// TIA Portal project "Perron038 AMR Siemens" (V14)

(* hardware
DEVICE "S7-1200 station_1"  S7-1200 Station
   slot 0: "Rack_0"  S7-1200 Rack  Rack  V1.0
   slot 1: "PLC_1"  CPU 1215C DC/DC/DC  6ES7 215-1AG40-0XB0  V4.2
*)

// ===== PLC "PLC_1"  CPU 1215C DC/DC/DC =====

VAR_GLOBAL   // PLC tag table "Default tag table"
   "Tag_1" AT %QW1000 : Word;
   "o_Output2" AT %Q0.1 : Bool;
   "Axis_1_Pulse" AT %Q0.0 : Bool;
   "M_stepEnable" AT %I0.0 : Bool;
   "q_driveEn" AT %Q0.2 : Bool;
   "q_stepOff" AT %Q0.3 : Bool;
   "M_ResetAxis" AT %I0.1 : Bool;
   "Jog_For" AT %I0.2 : Bool;
   "Jog_BWD" AT %I0.3 : Bool;
END_VAR

DATA_BLOCK "mainLogic_DB"   // DB1
{ S7_Optimized_Access := 'TRUE' }
VERSION : 0.1
// stored: InstanceOfName mainLogic
"mainLogic"
BEGIN
END_DATA_BLOCK

DATA_BLOCK "Axis_1"   // DB3, Motion_DB
{ S7_Optimized_Access := 'TRUE' }
AUTHOR : SIMATIC
FAMILY : BasicMC
NAME : TO_PosAx
VERSION : 6.0
// stored: InstanceOfName TO_PositioningAxis
"TO_PositioningAxis"
BEGIN
   // Axis.EnableOutput_AddressCU = %Q0.2
   // Axis.OnlinePtoModeCUEnumValue = PTO (pulse A and direction B)
   // Axis.OnlinePtoModeCU = 16#0000_0002
   // Axis.DirectionOutputEnabledCU = TRUE
   // Axis.SelectedChannel2EnumCU = %Q0.1
   // Axis.SelectedChannel1EnumCU = %Q0.0
   // Pulse.MinDeltaDeltaFrequencyCU = 0.004
   // Pulse.MaxDeltaDeltaFrequencyCU = 1.0E+10
   // Pulse.MinDeltaFrequencyCU = 0.005
   // Pulse.MaxDeltaFrequencyCU = 9.5E+9
   // Pulse.MinFrequencyCU = 1.0
   // Pulse.MaxFrequencyCU = 100000.0
   // Pulse.OutputSourceCU = 16#0000_0000
   // Axis.SelectPTO = 0
END_DATA_BLOCK

FUNCTION_BLOCK "mainLogic"   // FB1, SCL
{ S7_Optimized_Access := 'TRUE' }
VERSION : 0.1
   VAR_INPUT
      i_Input1 : Bool;
      i_Input2 : Bool;
   END_VAR
   VAR_OUTPUT
      q_Output1 : Bool;
      q_Output2 : Bool;
   END_VAR
BEGIN
       (* IF #i_Input1 THEN *)
           "Tag_1" := 70;
           #q_Output1 := 1;
           #q_Output2 := 1;
   (*    ELSIF #i_Input2 THEN
           #q_Output1 := 1;
           "Tag_1" := 30;
           #q_Output2 := 1;
       ELSE
           #q_Output1 := 1;
           "Tag_1" := 50;
           #q_Output2 := 0;
       END_IF;
       *)
END_FUNCTION_BLOCK

ORGANIZATION_BLOCK "Main"   // OB1, LAD, ProgramCycle
TITLE = "Main Program Sweep (Cycle)"
{ S7_Optimized_Access := 'TRUE' }
VERSION : 0.1
   VAR_INPUT
      Initial_Call : Bool;   // Initial call of this OB
      Remanence : Bool;   // =True, if remanent data are available
   END_VAR
   VAR_TEMP
      PWM_EN_1 : Bool;
   END_VAR
BEGIN

REGION Network 1: Initial call of this OB
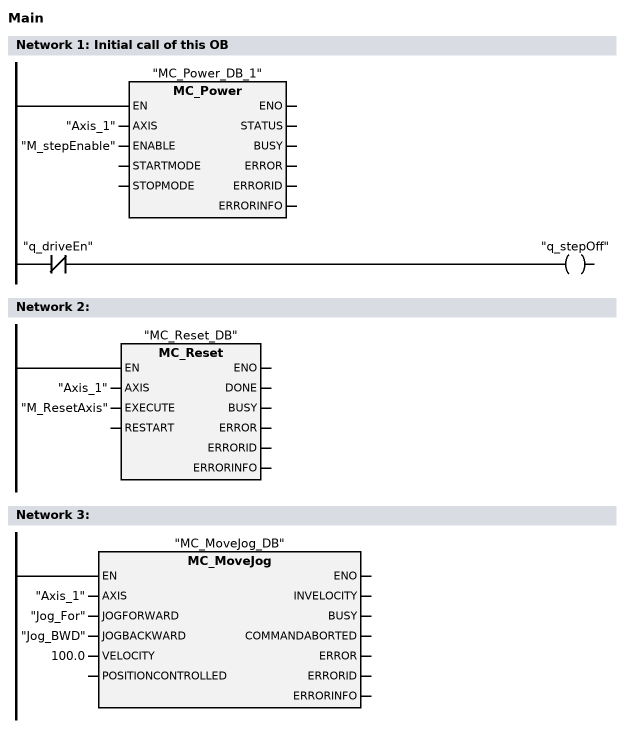
   "MC_Power_DB_1"(Axis := "Axis_1", Enable := "M_stepEnable");   // MC_Power
   "q_stepOff" := NOT "q_driveEn";
END_REGION

REGION Network 2
   "MC_Reset_DB"(Axis := "Axis_1", Execute := "M_ResetAxis");   // MC_Reset
END_REGION

REGION Network 3
   "MC_MoveJog_DB"(Axis := "Axis_1", JogForward := "Jog_For", JogBackward := "Jog_BWD", Velocity := 100.0);   // MC_MoveJog
END_REGION
END_ORGANIZATION_BLOCK